% RSLogix 500 project LAB2_BAW_BAK010.RSS, saved by version 8.40.00.08 %
PROJECT "LAB1_BAW"    % processor: SLC 500, 1747-L542 %

PROGRAM FILES
  LAD 2   37 rungs

DATA FILES
  O0 OUTPUT  68 elements
  I1 INPUT  68 elements
  S2 STATUS  164 elements
  B3 BINARY  9 elements
  T4 TIMER  34 elements
  C5 COUNTER  35 elements
  R6 CONTROL  1 elements
  N7 INTEGER  1 elements
  F8 FLOAT  1 elements

LADDER 2
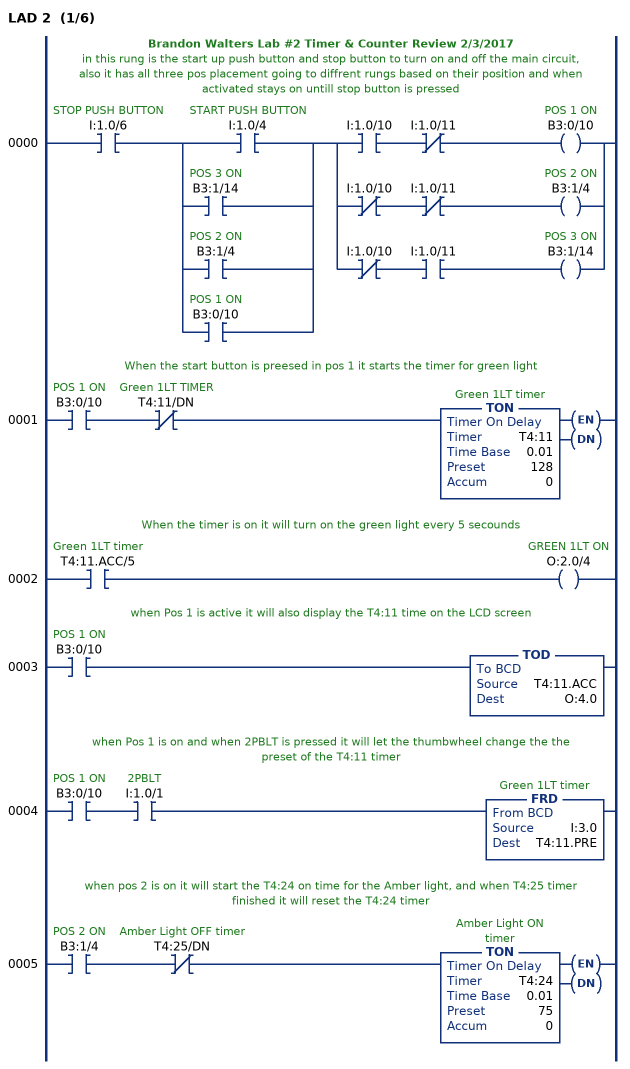
% Rung: 0 %
% TITLE: Brandon Walters Lab #2 Timer & Counter Review 2/3/2017 %
% in this rung is the start up push button and stop button to turn on and off the main circuit, also it has all three pos placement going to diffrent rungs based on their position and when activated stays on untill stop button is pressed %
SOR XIC I:1.0/6 BST XIC I:1.0/4 NXB XIC B3:1/14 NXB XIC B3:1/4 NXB XIC B3:0/10 BND BST XIC I:1.0/10 XIO I:1.0/11 OTE B3:0/10 NXB XIO I:1.0/10 XIO I:1.0/11 OTE B3:1/4 NXB XIO I:1.0/10 XIC I:1.0/11 OTE B3:1/14 BND EOR
%   I:1.0/6  "STOP PUSH BUTTON" %
%   I:1.0/4  "START PUSH BUTTON" %
%   B3:1/14  "POS 3 ON" %
%   B3:1/4  "POS 2 ON" %
%   B3:0/10  "POS 1 ON" %
% Rung: 1 %
% When the start button is preesed in pos 1 it starts the timer for green light %
SOR XIC B3:0/10 XIO T4:11/DN TON T4:11 0.01 128 0 EOR
%   B3:0/10  "POS 1 ON" %
%   T4:11/DN  "Green 1LT TIMER" %
%   T4:11  "Green 1LT timer" %
% Rung: 2 %
% When the timer is on it will turn on the green light every 5 secounds %
SOR XIC T4:11.ACC/5 OTE O:2.0/4 EOR
%   T4:11  "Green 1LT timer" %
%   O:2.0/4  "GREEN 1LT ON" %
% Rung: 3 %
% when Pos 1 is active it will also display the T4:11 time on the LCD screen %
SOR XIC B3:0/10 TOD T4:11.ACC O:4.0 EOR
%   B3:0/10  "POS 1 ON" %
%   T4:11  "Green 1LT timer" %
% Rung: 4 %
% when Pos 1 is on and when 2PBLT is pressed it will let the thumbwheel change the the preset of the T4:11 timer %
SOR XIC B3:0/10 XIC I:1.0/1 FRD I:3.0 T4:11.PRE EOR
%   B3:0/10  "POS 1 ON" %
%   I:1.0/1  "2PBLT" %
%   I:3.0  "RED TOWER TIME DISPLAY" %
%   T4:11  "Green 1LT timer" %
% Rung: 5 %
% when pos 2 is on it will start the T4:24 on time for the Amber light, and when T4:25 timer finished it will reset the T4:24 timer %
SOR XIC B3:1/4 XIO T4:25/DN TON T4:24 0.01 75 0 EOR
%   B3:1/4  "POS 2 ON" %
%   T4:25  "Amber Light OFF timer" %
%   T4:24  "Amber Light ON timer" %

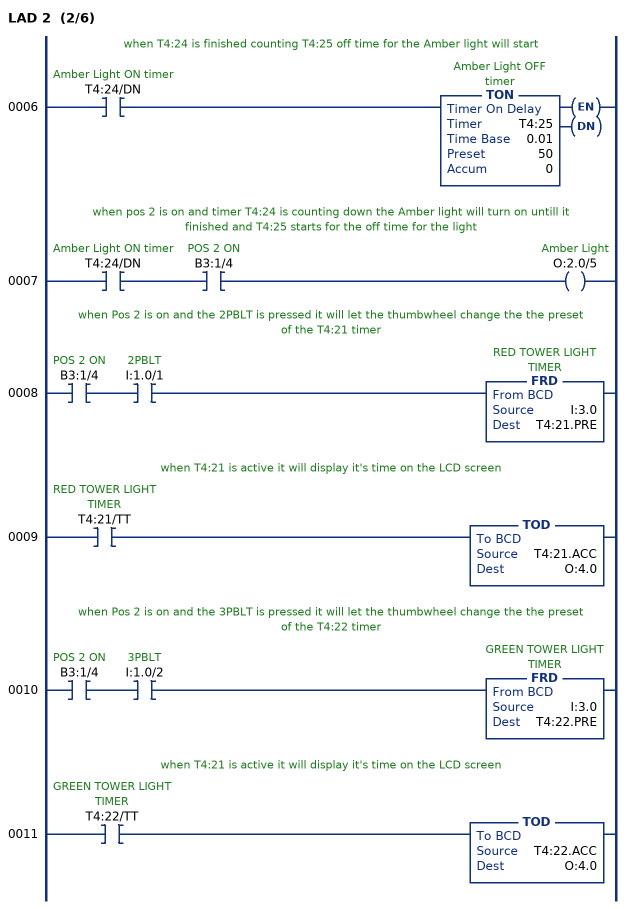
% Rung: 6 %
% when T4:24 is finished counting T4:25 off time for the Amber light will start %
SOR XIC T4:24/DN TON T4:25 0.01 50 0 EOR
%   T4:24  "Amber Light ON timer" %
%   T4:25  "Amber Light OFF timer" %
% Rung: 7 %
% when pos 2 is on and timer T4:24 is counting down the Amber light will turn on untill it finished and T4:25 starts for the off time for the light %
SOR XIC T4:24/DN XIC B3:1/4 OTE O:2.0/5 EOR
%   T4:24  "Amber Light ON timer" %
%   B3:1/4  "POS 2 ON" %
%   O:2.0/5  "Amber Light" %
% Rung: 8 %
% when Pos 2 is on and the 2PBLT is pressed it will let the thumbwheel change the the preset of the T4:21 timer %
SOR XIC B3:1/4 XIC I:1.0/1 FRD I:3.0 T4:21.PRE EOR
%   B3:1/4  "POS 2 ON" %
%   I:1.0/1  "2PBLT" %
%   I:3.0  "RED TOWER TIME DISPLAY" %
%   T4:21  "RED TOWER LIGHT TIMER" %
% Rung: 9 %
% when T4:21 is active it will display it's time on the LCD screen %
SOR XIC T4:21/TT TOD T4:21.ACC O:4.0 EOR
%   T4:21  "RED TOWER LIGHT TIMER" %
% Rung: 10 %
% when Pos 2 is on and the 3PBLT is pressed it will let the thumbwheel change the the preset of the T4:22 timer %
SOR XIC B3:1/4 XIC I:1.0/2 FRD I:3.0 T4:22.PRE EOR
%   B3:1/4  "POS 2 ON" %
%   I:1.0/2  "3PBLT" %
%   I:3.0  "RED TOWER TIME DISPLAY" %
%   T4:22  "GREEN TOWER LIGHT TIMER" %
% Rung: 11 %
% when T4:21 is active it will display it's time on the LCD screen %
SOR XIC T4:22/TT TOD T4:22.ACC O:4.0 EOR
%   T4:22  "GREEN TOWER LIGHT TIMER" %

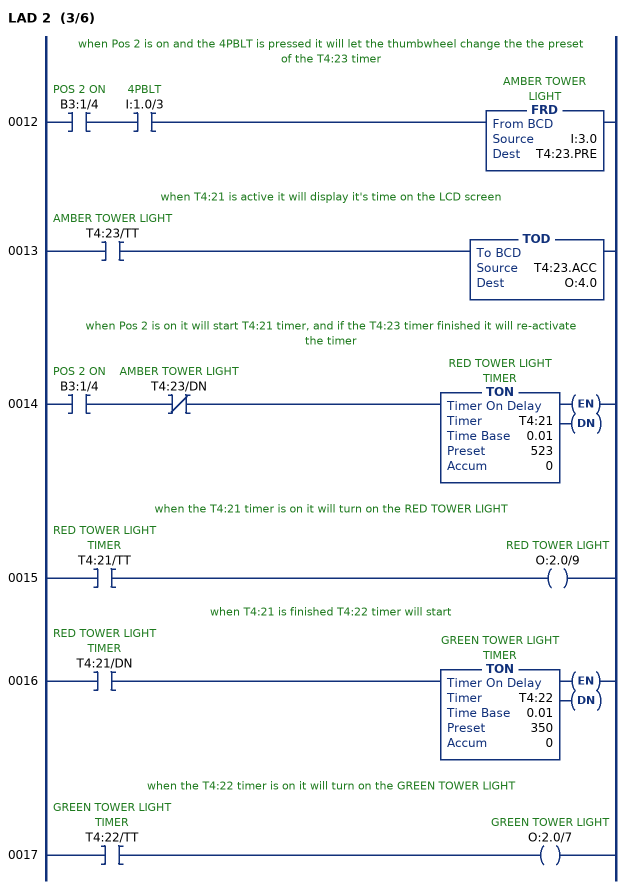
% Rung: 12 %
% when Pos 2 is on and the 4PBLT is pressed it will let the thumbwheel change the the preset of the T4:23 timer %
SOR XIC B3:1/4 XIC I:1.0/3 FRD I:3.0 T4:23.PRE EOR
%   B3:1/4  "POS 2 ON" %
%   I:1.0/3  "4PBLT" %
%   I:3.0  "RED TOWER TIME DISPLAY" %
%   T4:23  "AMBER TOWER LIGHT" %
% Rung: 13 %
% when T4:21 is active it will display it's time on the LCD screen %
SOR XIC T4:23/TT TOD T4:23.ACC O:4.0 EOR
%   T4:23  "AMBER TOWER LIGHT" %
% Rung: 14 %
% when Pos 2 is on it will start T4:21 timer, and if the T4:23 timer finished it will re-activate the timer %
SOR XIC B3:1/4 XIO T4:23/DN TON T4:21 0.01 523 0 EOR
%   B3:1/4  "POS 2 ON" %
%   T4:23  "AMBER TOWER LIGHT" %
%   T4:21  "RED TOWER LIGHT TIMER" %
% Rung: 15 %
% when the T4:21 timer is on it will turn on the RED TOWER LIGHT %
SOR XIC T4:21/TT OTE O:2.0/9 EOR
%   T4:21  "RED TOWER LIGHT TIMER" %
%   O:2.0/9  "RED TOWER LIGHT" %
% Rung: 16 %
% when T4:21 is finished T4:22 timer will start %
SOR XIC T4:21/DN TON T4:22 0.01 350 0 EOR
%   T4:21  "RED TOWER LIGHT TIMER" %
%   T4:22  "GREEN TOWER LIGHT TIMER" %
% Rung: 17 %
% when the T4:22 timer is on it will turn on the GREEN TOWER LIGHT %
SOR XIC T4:22/TT OTE O:2.0/7 EOR
%   T4:22  "GREEN TOWER LIGHT TIMER" %
%   O:2.0/7  "GREEN TOWER LIGHT" %

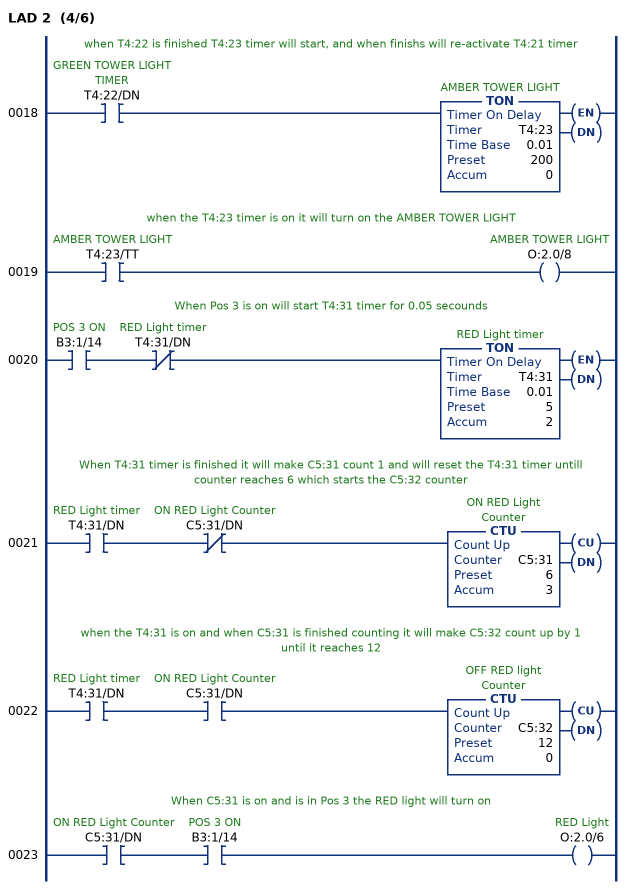
% Rung: 18 %
% when T4:22 is finished T4:23 timer will start, and when finishs will re-activate T4:21 timer %
SOR XIC T4:22/DN TON T4:23 0.01 200 0 EOR
%   T4:22  "GREEN TOWER LIGHT TIMER" %
%   T4:23  "AMBER TOWER LIGHT" %
% Rung: 19 %
% when the T4:23 timer is on it will turn on the AMBER TOWER LIGHT %
SOR XIC T4:23/TT OTE O:2.0/8 EOR
%   T4:23  "AMBER TOWER LIGHT" %
%   O:2.0/8  "AMBER TOWER LIGHT" %
% Rung: 20 %
% When Pos 3 is on will start T4:31 timer for 0.05 secounds %
SOR XIC B3:1/14 XIO T4:31/DN TON T4:31 0.01 5 2 EOR
%   B3:1/14  "POS 3 ON" %
%   T4:31  "RED Light timer" %
% Rung: 21 %
% When T4:31 timer is finished it will make C5:31 count 1 and will reset the T4:31 timer untill counter reaches 6 which starts the C5:32 counter %
SOR XIC T4:31/DN XIO C5:31/DN CTU C5:31 6 3 EOR
%   T4:31  "RED Light timer" %
%   C5:31  "ON RED Light Counter" %
% Rung: 22 %
% when the T4:31 is on and when C5:31 is finished counting it will make C5:32 count up by 1 until it reaches 12 %
SOR XIC T4:31/DN XIC C5:31/DN CTU C5:32 12 0 EOR
%   T4:31  "RED Light timer" %
%   C5:31  "ON RED Light Counter" %
%   C5:32  "OFF RED light Counter" %
% Rung: 23 %
% When C5:31 is on and is in Pos 3 the RED light will turn on %
SOR XIC C5:31/DN XIC B3:1/14 OTE O:2.0/6 EOR
%   C5:31  "ON RED Light Counter" %
%   B3:1/14  "POS 3 ON" %
%   O:2.0/6  "RED Light" %

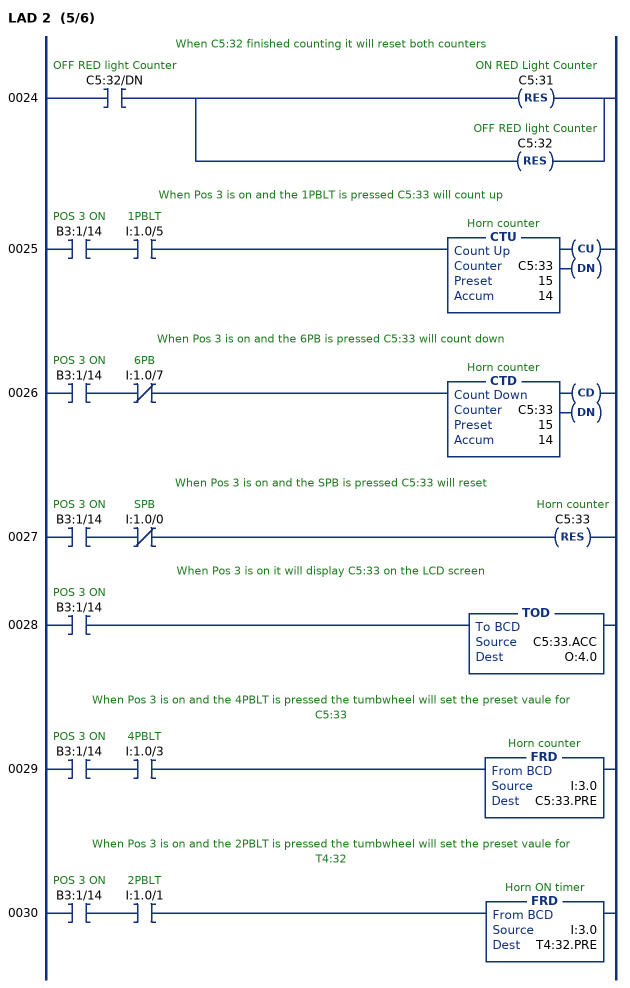
% Rung: 24 %
% When C5:32 finished counting it will reset both counters %
SOR XIC C5:32/DN BST RES C5:31 NXB RES C5:32 BND EOR
%   C5:32  "OFF RED light Counter" %
%   C5:31  "ON RED Light Counter" %
% Rung: 25 %
% When Pos 3 is on and the 1PBLT is pressed C5:33 will count up %
SOR XIC B3:1/14 XIC I:1.0/5 CTU C5:33 15 14 EOR
%   B3:1/14  "POS 3 ON" %
%   I:1.0/5  "1PBLT" %
%   C5:33  "Horn counter" %
% Rung: 26 %
% When Pos 3 is on and the 6PB is pressed C5:33 will count down %
SOR XIC B3:1/14 XIO I:1.0/7 CTD C5:33 15 14 EOR
%   B3:1/14  "POS 3 ON" %
%   I:1.0/7  "6PB" %
%   C5:33  "Horn counter" %
% Rung: 27 %
% When Pos 3 is on and the SPB is pressed C5:33 will reset %
SOR XIC B3:1/14 XIO I:1.0/0 RES C5:33 EOR
%   B3:1/14  "POS 3 ON" %
%   I:1.0/0  "SPB" %
%   C5:33  "Horn counter" %
%   RES C5:33  "COUNTER RESET" %
% Rung: 28 %
% When Pos 3 is on it will display C5:33 on the LCD screen %
SOR XIC B3:1/14 TOD C5:33.ACC O:4.0 EOR
%   B3:1/14  "POS 3 ON" %
%   C5:33  "Horn counter" %
% Rung: 29 %
% When Pos 3 is on and the 4PBLT is pressed the tumbwheel will set the preset vaule for C5:33 %
SOR XIC B3:1/14 XIC I:1.0/3 FRD I:3.0 C5:33.PRE EOR
%   B3:1/14  "POS 3 ON" %
%   I:1.0/3  "4PBLT" %
%   I:3.0  "RED TOWER TIME DISPLAY" %
%   C5:33  "Horn counter" %
% Rung: 30 %
% When Pos 3 is on and the 2PBLT is pressed the tumbwheel will set the preset vaule for T4:32 %
SOR XIC B3:1/14 XIC I:1.0/1 FRD I:3.0 T4:32.PRE EOR
%   B3:1/14  "POS 3 ON" %
%   I:1.0/1  "2PBLT" %
%   I:3.0  "RED TOWER TIME DISPLAY" %
%   T4:32  "Horn ON timer" %

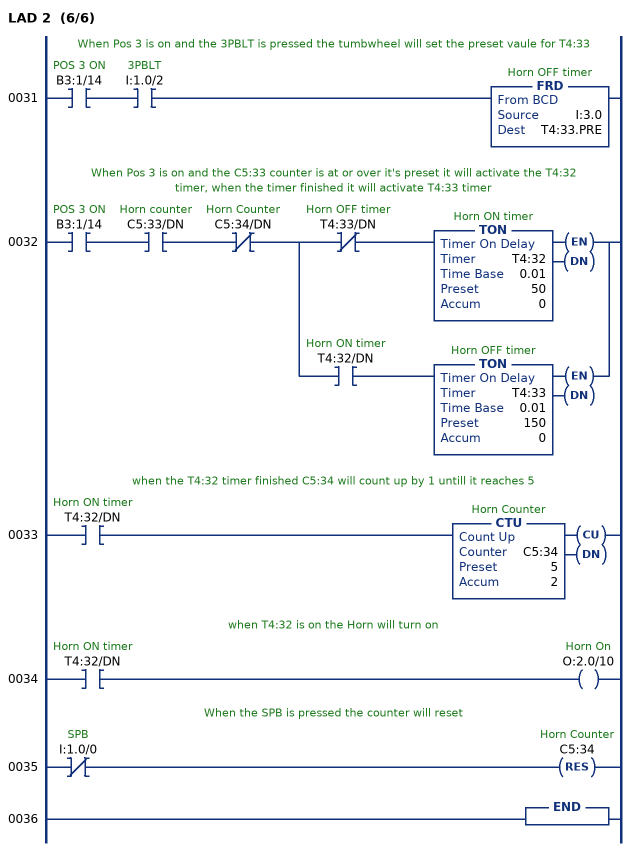
% Rung: 31 %
% When Pos 3 is on and the 3PBLT is pressed the tumbwheel will set the preset vaule for T4:33 %
SOR XIC B3:1/14 XIC I:1.0/2 FRD I:3.0 T4:33.PRE EOR
%   B3:1/14  "POS 3 ON" %
%   I:1.0/2  "3PBLT" %
%   I:3.0  "RED TOWER TIME DISPLAY" %
%   T4:33  "Horn OFF timer" %
% Rung: 32 %
% When Pos 3 is on and the C5:33 counter is at or over it's preset it will activate the T4:32 timer, when the timer finished it will activate T4:33 timer %
SOR XIC B3:1/14 XIC C5:33/DN XIO C5:34/DN BST XIO T4:33/DN TON T4:32 0.01 50 0 NXB XIC T4:32/DN TON T4:33 0.01 150 0 BND EOR
%   B3:1/14  "POS 3 ON" %
%   C5:33  "Horn counter" %
%   C5:34  "Horn Counter" %
%   T4:33  "Horn OFF timer" %
%   T4:32  "Horn ON timer" %
% Rung: 33 %
% when the T4:32 timer finished C5:34 will count up by 1 untill it reaches 5 %
SOR XIC T4:32/DN CTU C5:34 5 2 EOR
%   T4:32  "Horn ON timer" %
%   C5:34  "Horn Counter" %
% Rung: 34 %
% when T4:32 is on the Horn will turn on %
SOR XIC T4:32/DN OTE O:2.0/10 EOR
%   T4:32  "Horn ON timer" %
%   O:2.0/10  "Horn On" %
% Rung: 35 %
% When the SPB is pressed the counter will reset %
SOR XIO I:1.0/0 RES C5:34 EOR
%   I:1.0/0  "SPB" %
%   C5:34  "Horn Counter" %
% Rung: 36 %
SOR END EOR

COMMENTS NOT ATTACHED TO A CURRENT RUNG
  C5:33: When Pos 3 is on and the 2PBLT is pressed C5:33 will count up

REVISION NOTES
  0: connected

DATA TABLE (non-zero values as saved)
DATA B3
% B3:0 % 0X0000 0X4000 0X0000 0X0000 0X0000 0X0000 0X0000 0X0000 0X0000
DATA T4
% .PRE .ACC %
% T4:1 % 32 1
% T4:2 % 32 1
% T4:11 % 128 0
% T4:21 % 523 0
% T4:22 % 350 0
% T4:23 % 200 0
% T4:24 % 75 0
% T4:25 % 50 0
% T4:31 % 5 2
% T4:32 % 50 0
% T4:33 % 150 0
DATA C5
% .PRE .ACC %
% C5:31 % 6 3
% C5:32 % 12 0
% C5:33 % 15 14
% C5:34 % 5 2
